Universal Robots PolyScope program: demo sleeve fillet 2.urp

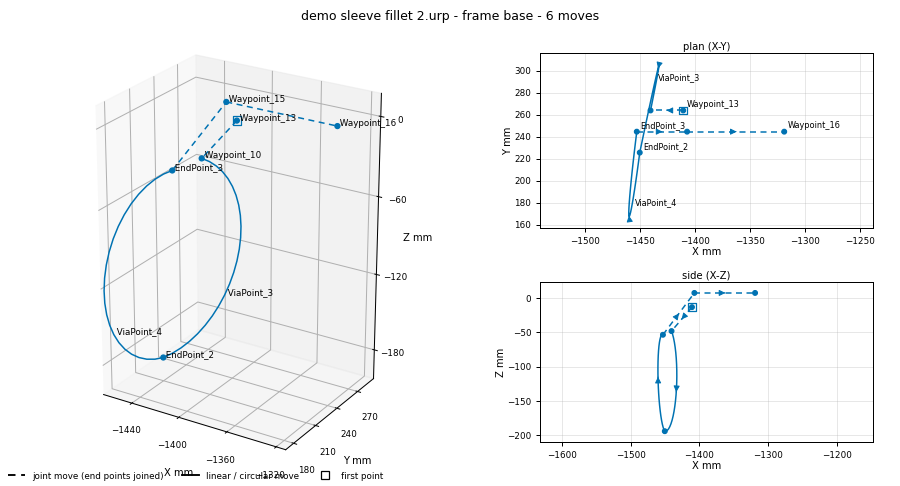
[picture p0: tool path of demo sleeve fillet 2.urp in frame base, 6 of 8 moves have a stored position in this frame; points joined in program order, loops and branches not executed]
Program demo sleeve fillet 2 (installation=default directory=/programs createdIn=5.21.3 lastSavedIn=5.21.3 robotSerialNumber=20246801938)
Calibrated DH parameters: a=[-0.000071, -0.790281, -0.600694, 0.000061, -0.000039, 0]; d=[0.236272, 604.465945, 132.116513, -736.382239, 0.159268, 0.154005]; alpha=[1.570254, -0.000567, 0.000559, 1.571709, -1.56999, 0]; deltaTheta=[0, -0.409357, 7.293326, -0.600784, -0.000001, -0.000001]
InitVariablesNode
Robot Program (runOnlyOnce=false)
  Set NoAction tcp=pretend_welder
  SuppressedNode
    MoveJ speed 60 deg/s, acceleration 80 deg/s^2 (useActiveTCP=true optimoveEnabled=false optiMoveSpeed=0.3 optiMoveAcceleration=0.09) feature=Base
      SuppressedNode
        Waypoint Waypoint_3: TCP in base x=-912.453 y=673.518 z=718.985 mm, rx=-0.4706 ry=-1.9428 rz=0.4955 rad; joints [-63.285, -68.284, 110.161, 88.985, -83.541, -118.353] deg; TCP offset x=-9.5 y=-328 z=105.73 mm, rx=1.2092 ry=-1.2092 rz=1.2092 rad
      SuppressedNode
        Waypoint Waypoint_4: TCP in base x=-1043.534 y=752.126 z=758.241 mm, rx=-0.4498 ry=-2.3257 rz=-0.2665 rad; joints [-53.991, -67.414, 94.218, 102.936, -66.691, -159.337] deg
      Waypoint Waypoint_9: TCP in base x=-850.146 y=808.476 z=769.845 mm, rx=-0.0694 ry=-2.4231 rz=-0.6317 rad; joints [-70.02, -72.001, 93.194, -274.04, -37.901, -142.904] deg
      Waypoint Waypoint_6: TCP in base x=-1042.273 y=808.476 z=769.845 mm, rx=-0.0694 ry=-2.4231 rz=-0.6317 rad; joints [-58.413, -64.349, 84.656, -260.501, -42.539, -159.423] deg
  SuppressedNode
    MoveJ speed 60 deg/s, acceleration 80 deg/s^2 (useActiveTCP=true optimoveEnabled=false optiMoveSpeed=0.3 optiMoveAcceleration=0.09) feature=Base
      SuppressedNode
        Waypoint Waypoint_1: TCP in base x=-1152.594 y=814.679 z=699.964 mm, rx=0.098 ry=-2.3843 rz=-0.4483 rad; joints [-56.525, -54.403, 73.307, 93.455, -42.841, -145.624] deg
      SuppressedNode
        Waypoint Waypoint_5: TCP in base x=-1149.758 y=814.958 z=702.794 mm, rx=-0.0472 ry=-2.3472 rz=-0.7271 rad; joints [-53.278, -57.004, 80.845, -264.711, -44.526, -166.31] deg
      Waypoint Waypoint_7: TCP in base x=-1150.142 y=824.468 z=703.476 mm, rx=-0.1355 ry=-2.1954 rz=-0.513 rad; joints [-54.373, -54.473, 80.141, -274.253, -56.089, -154.835] deg
  SuppressedNode
    MoveP speed 10 mm/s, acceleration 1200 mm/s^2 (blendRadius=0.025 useActiveTCP=true optimoveEnabled=false optiMoveSpeed=0.3 optiMoveAcceleration=0.09) feature=Base
      CircleMove (OrientationMode=FIXED)
        Waypoint ViaPoint_1: TCP in base x=-1137.967 y=888.777 z=671.431 mm, rx=-0.7156 ry=-2.1833 rz=0.6859 rad; joints [-57.632, -55.198, 82.444, 124.608, -82.298, -128.207] deg
        Waypoint EndPoint_1: TCP in base x=-1139.924 y=872.884 z=596.072 mm, rx=-1.219 ry=-0.9297 rz=2.3215 rad; joints [-60.159, -58.197, 98.87, 176.452, -78.393, -68.042] deg
      CircleMove (OrientationMode=FIXED)
        Waypoint ViaPoint_2: TCP in base x=-1155.211 y=763.52 z=646.144 mm, rx=0.9307 ry=-1.6945 rz=-2.1414 rad; joints [-52.747, -75.971, 108.96, 234.472, -18.82, -4.377] deg
        Waypoint Waypoint_1: TCP in base x=-1152.594 y=814.679 z=699.964 mm, rx=0.098 ry=-2.3843 rz=-0.4483 rad; joints [-56.525, -54.403, 73.307, 93.455, -42.841, -145.624] deg
  SuppressedNode
    MoveJ speed 60 deg/s, acceleration 80 deg/s^2 (useActiveTCP=true optimoveEnabled=false optiMoveSpeed=0.3 optiMoveAcceleration=0.09) feature=Base
      SuppressedNode
        Waypoint Waypoint_2: TCP in base x=-917.75 y=830.261 z=524.512 mm, rx=-1.543 ry=-0.8444 rz=1.9881 rad; joints [-66.08, -72.484, 118.808, 175.962, -93.351, -73.55] deg
      Waypoint Waypoint_4: TCP in base x=-1043.534 y=752.126 z=758.241 mm, rx=-0.4498 ry=-2.3257 rz=-0.2665 rad; joints [-53.991, -67.414, 94.218, 102.936, -66.691, -159.337] deg
      Waypoint Waypoint_8: TCP in base x=-754.583 y=757.082 z=772.781 mm, rx=-0.4498 ry=-2.3257 rz=-0.2665 rad; joints [-73.782, -79.343, 107.572, 92.439, -55.198, -140.846] deg
  SuppressedNode
    Folder half circle
      MoveJ speed 60 deg/s, acceleration 80 deg/s^2 (useActiveTCP=true optimoveEnabled=false optiMoveSpeed=0.3 optiMoveAcceleration=0.09) feature=Base
        Waypoint Waypoint_13: TCP in base x=-1410.884 y=263.861 z=-13.194 mm, rx=-0.2057 ry=-2.2742 rz=-0.4378 rad; joints [-18.611, -21.126, 85.064, -293.08, -78.09, -188.172] deg
      MoveJ speed 60 deg/s, acceleration 80 deg/s^2 (useActiveTCP=true optimoveEnabled=false optiMoveSpeed=0.3 optiMoveAcceleration=0.09) feature=Base
        Waypoint Waypoint_10: TCP in base x=-1440.647 y=263.861 z=-48.062 mm, rx=-0.2057 ry=-2.2742 rz=-0.4378 rad; joints [-18.086, -18.126, 80.761, -291.695, -78.433, -188.577] deg
        SuppressedNode
          Waypoint Waypoint_11: TCP in base x=-1286.175 y=549.195 z=115.468 mm, rx=-0.27 ry=-1.5277 rz=-1.42 rad; joints [-20.499, -22.138, 88.563, -259.74, -128.557, -138.212] deg; TCP offset x=-1.032 y=-18.062 z=285.234 mm, rx=0 ry=0 rz=0 rad
        SuppressedNode
          Waypoint Waypoint_12: TCP in base x=-1198.19 y=495.746 z=-342.486 mm, rx=-1.4417 ry=-1.7142 rz=-0.5215 rad; joints [-20.358, -19.189, 100.698, -215.464, -126.338, -45.331] deg
      MoveP speed 8 mm/s, acceleration 1200 mm/s^2 (blendRadius=0.025 useActiveTCP=true optimoveEnabled=false optiMoveSpeed=0.3 optiMoveAcceleration=0.09) feature=Base
        CircleMove (OrientationMode=FIXED)
          Waypoint ViaPoint_3: TCP in base x=-1436.982 y=288.423 z=-164.849 mm, rx=-1.2985 ry=-1.3493 rz=1.8084 rad; joints [-22.4, -18.108, 96.782, -229.781, -128.579, -68.735] deg; TCP offset x=-9.5 y=-328 z=105.73 mm, rx=1.2092 ry=-1.2092 rz=1.2092 rad
          Waypoint EndPoint_2: TCP in base x=-1450.471 y=225.502 z=-193.907 mm, rx=-1.3296 ry=-0.3697 rz=2.6077 rad; joints [-22.267, -13.945, 97.987, -213.988, -92.35, -25.678] deg
      MoveJ speed 60 deg/s, acceleration 80 deg/s^2 (useActiveTCP=true optimoveEnabled=false optiMoveSpeed=0.3 optiMoveAcceleration=0.09) feature=Base
        Waypoint Waypoint_14: TCP in base x=-1380.88 y=218.821 z=-252.804 mm, rx=-1.3435 ry=-0.3935 rz=2.6113 rad; joints [-23.838, -10.524, 100.952, -220.078, -91.217, -28.02] deg
  Folder full circle
    MoveJ speed 60 deg/s, acceleration 80 deg/s^2 (useActiveTCP=true optimoveEnabled=false optiMoveSpeed=0.3 optiMoveAcceleration=0.09) feature=Base
      Waypoint Waypoint_13: TCP in base x=-1410.884 y=263.861 z=-13.194 mm, rx=-0.2057 ry=-2.2742 rz=-0.4378 rad; joints [-18.611, -21.126, 85.064, -293.08, -78.09, -188.172] deg
    MoveJ speed 60 deg/s, acceleration 80 deg/s^2 (useActiveTCP=true optimoveEnabled=false optiMoveSpeed=0.3 optiMoveAcceleration=0.09) feature=Base
      Waypoint Waypoint_10: TCP in base x=-1440.647 y=263.861 z=-48.062 mm, rx=-0.2057 ry=-2.2742 rz=-0.4378 rad; joints [-18.086, -18.126, 80.761, -291.695, -78.433, -188.577] deg
      SuppressedNode
        Waypoint Waypoint_11: TCP in base x=-1286.175 y=549.195 z=115.468 mm, rx=-0.27 ry=-1.5277 rz=-1.42 rad; joints [-20.499, -22.138, 88.563, -259.74, -128.557, -138.212] deg; TCP offset x=-1.032 y=-18.062 z=285.234 mm, rx=0 ry=0 rz=0 rad
      SuppressedNode
        Waypoint Waypoint_12: TCP in base x=-1198.19 y=495.746 z=-342.486 mm, rx=-1.4417 ry=-1.7142 rz=-0.5215 rad; joints [-20.358, -19.189, 100.698, -215.464, -126.338, -45.331] deg
    MoveP speed 8 mm/s, acceleration 1200 mm/s^2 (blendRadius=0.025 useActiveTCP=true optimoveEnabled=false optiMoveSpeed=0.3 optiMoveAcceleration=0.09) feature=Base
      CircleMove (OrientationMode=FIXED)
        Waypoint ViaPoint_3: TCP in base x=-1436.982 y=288.423 z=-164.849 mm, rx=-1.2985 ry=-1.3493 rz=1.8084 rad; joints [-22.4, -18.108, 96.782, -229.781, -128.579, -68.735] deg; TCP offset x=-9.5 y=-328 z=105.73 mm, rx=1.2092 ry=-1.2092 rz=1.2092 rad
        Waypoint EndPoint_2: TCP in base x=-1450.471 y=225.502 z=-193.907 mm, rx=-1.3296 ry=-0.3697 rz=2.6077 rad; joints [-22.267, -13.945, 97.987, -213.988, -92.35, -25.678] deg
      CircleMove (OrientationMode=FIXED)
        Waypoint ViaPoint_4: TCP in base x=-1458.06 y=174.729 z=-155.961 mm, rx=0.9854 ry=-0.8297 rz=-2.4175 rad; joints [-21.89, -10.796, 94.59, -213.949, -40.159, 6.455] deg
        Waypoint EndPoint_3: TCP in base x=-1453.174 y=244.554 z=-53.456 mm, rx=-0.0081 ry=-2.2253 rz=-0.4366 rad; joints [-20.236, -35.116, 108.931, -127.571, 69.187, -2.082] deg
    MoveL speed 250 mm/s, acceleration 1200 mm/s^2 (useActiveTCP=true optimoveEnabled=false optiMoveSpeed=0.3 optiMoveAcceleration=0.09) feature=Base
      MoveDirectionNode expression=[1.0,0.0,1.0]
        Until DISTANCE (allowActions=false deceleration=3 distanceNodeType=STOP) Distance=0.1; motionParameters(blendRadius=0)
    MoveJ speed 60 deg/s, acceleration 80 deg/s^2 (useActiveTCP=true optimoveEnabled=false optiMoveSpeed=0.3 optiMoveAcceleration=0.09) feature=Base
      Waypoint Waypoint_15: TCP in base x=-1407.381 y=244.554 z=7.478 mm, rx=-0.0081 ry=-2.2253 rz=-0.4366 rad; joints [-21.148, -40.183, 113.996, -127.853, 68.651, -1.292] deg
      Waypoint Waypoint_16: TCP in base x=-1318.966 y=244.554 z=7.478 mm, rx=1.059 ry=-2.1109 rz=-0.921 rad; joints [-32.341, -42.763, 117.442, -171.905, 11.465, 43.721] deg
